{attribute addProperty BoxType "ELX1052-0000-0016"}
{attribute addProperty Id "ChannelAT %I*ARRAY[0..1] OF Channel_E18390663240WcStateAT %I*WcState_F855686C1620InfoDataAT %I*InfoData_192954DE1620"}
{attribute addProperty CRC "2090431803"}
{attribute addProperty SizeInBites "64"}
{attribute addProperty SizeInBytes "8"}
TYPE ELX1052_0A1DBF07 :
STRUCT
	{attribute addProperty Name "Channel"}
	Channel : ARRAY[0..1] OF Channel_E1839066;
	{attribute addProperty Name "WcState"}
	WcState : WcState_F855686C;
	{attribute addProperty Name "InfoData"}
	InfoData : InfoData_192954DE;
END_STRUCT
END_TYPE

(* stored: Version 1.2.0.0, ProductVersion 3.1.4024.9
   DUT ELX1052_0A1DBF07: Id {77454b88-2e38-4b3b-9097-aee0115e28a1} *)
